FUNCTION_BLOCK FB_Fahrlogik1
VAR_INPUT
END_VAR
VAR_OUTPUT
END_VAR
VAR
END_VAR

END_FUNCTION_BLOCK

(* stored: Version 1.1.0.1
   POU FB_Fahrlogik1: Id {f31a1d73-9b92-45fa-998d-d2a6ec7ce41c}, SpecialFunc None *)
